// TwinCAT 3 PLC project Untitled1
// ProgramVersion: 3.1.4024.0
// libraries:
//   Tc2_Standard, * (Beckhoff Automation GmbH)
//   Tc2_System, * (Beckhoff Automation GmbH)
//   Tc3_Module, * (Beckhoff Automation GmbH)
//   VisuDialogs, * (System)
//   VisuSymbols,3.5.10.0,System
// project tree:
//   / DUT.TcDUT, GlobalTextList.TcGTLO, Param.TcGVL, PlcTask.TcTTO, Visualization Manager.TcVMO (not stored)
//   DUTs/ weekDays.TcDUT
//   GVLs/ GVL.TcGVL
//   POUs/ MAIN.TcPOU, Routine1.TcPOU, Routine2.TcPOU
//   VISUs/ Visualization.TcVIS
// real-time tasks:
//   TASK PlcTask: cycle T#10ms, priority 20, ADS port 350

CONFIGURATION Untitled1
    RESOURCE PLC ON TwinCAT3
        TASK PlcTask(INTERVAL := T#10ms, PRIORITY := 20);
        PROGRAM MAIN WITH PlcTask : MAIN;
    END_RESOURCE
END_CONFIGURATION

// ---- DUT.TcDUT
TYPE DUT :
STRUCT
END_STRUCT
END_TYPE

// ---- DUTs/weekDays.TcDUT
TYPE weekDays :
STRUCT
	Mon : STRING;
	Tue : STRING;
	Wend: STRING;
	Thu	: STRING;
	Fri	: STRING;
	
END_STRUCT
END_TYPE

// ---- GVLs/GVL.TcGVL
{attribute 'qualified_only'}
VAR_GLOBAL
	Morning 		: BOOL := FALSE	 ;
	
	WakeUp			: BOOL	 ;
	DateCheck		: BOOL	 ;
	ComeBackHome	: BOOL	 ;
	TakeShower		: BOOL	 ;
	GoToBed			: BOOL 	 ;
	MakeTheBed		: BOOL   ;
	MakeCoffee		: BOOL	 ;
	EatBreakfast	: BOOL	 ;
	Day 			: STRING ;
	Routine1 		: BOOL 	 ;
	Routine2		: BOOL	 ;
	
	
			
END_VAR

// ---- Param.TcGVL
{attribute 'qualified_only'}
VAR_GLOBAL CONSTANT
END_VAR

// ---- POUs/MAIN.TcPOU
PROGRAM MAIN
VAR
	State 			: INT	:= 5 ;

	ToTimeoutbool 	: TON ;
	T1Timer 		: BOOL ;
	enable 			: BOOL;
	rTrigenable 	: R_TRIG;
	
END_VAR

rTrigenable(CLk := enable);
ToTimeoutbool(IN := T1Timer,PT := T#2S);
IF gvl.Morning THEN
	state := 0;
END_IF
	CASE state OF
	0:
		GVL.WakeUp 					:= TRUE;
		T1Timer 					:= TRUE;
		IF ToTimeoutbool.Q THEN
			T1Timer 				:= FALSE;
			GVL.WakeUp 				:= FALSE ;
			state := 1; 
		END_IF
		
	1:
		GVL.MakeTheBed 				:= TRUE;
			T1Timer 				:= TRUE;
		IF ToTimeoutbool.Q THEN
			T1Timer 				:= FALSE;
			GVL.MakeTheBed 			:= FALSE ;
			state := 2;
		END_IF
		
	2:
		GVL.TakeShower 				:= TRUE;
		T1Timer 					:= TRUE;
		IF ToTimeoutbool.Q THEN
			T1Timer := FALSE;
			GVL.TakeShower 			:= FALSE ;
			state := 3;
		END_IF
		
	3:
		GVL.DateCheck				:= TRUE;
		State := 4; 

	4: 
		IF gvl.Day = 'Sat' OR gvl.Day = 'Sun' THEN
			routine2();
			gvl.Routine2 			:= TRUE;
			
		ELSIF gvl.Day = 'Fri' OR gvl.Day = 'Mon' OR gvl.Day = 'Tue' OR gvl.Day = 'Wend' OR gvl.Day = 'Thu' THEN
		 	routine1();		
			GVl.Routine1 			:= TRUE ;
			
		END_IF
	
		
	END_CASE

END_PROGRAM

// ---- POUs/Routine2.TcPOU
PROGRAM Routine2
VAR
	     
	DoLaundriesR2             	: BOOL ; 
	DoGroceriesR2            	: BOOL ; 
	
	OrganizeGroceriesR2      	: BOOL ; 
	CheckWashingMachineR2    	: BOOL ; 
	DoOtherChoresR2         	: BOOL ; 
	CookSomethingR2           	: BOOL ; 
	UnloadMachineR2          	: BOOL ;  
	EatLunchR2					: BOOL ;
	State 						: INT :=0  ;
	Day  						: STRING  ;
	ToTimeoutbool 				: TON ;
	T1Timer 					: BOOL ;
	enable 						: BOOL;
	rTrigenable 				: R_TRIG;
END_VAR

rTrigenable(CLk := enable);
ToTimeoutbool(IN := T1Timer,PT := T#2S);
gvl.DateCheck := FALSE ;

CASE state OF
	0:
		GVL.MakeCoffee 					:= TRUE;
		T1Timer 						:= TRUE;
		IF ToTimeoutbool.Q THEN
			T1Timer 					:= FALSE;
			GVL.MakeCoffee 				:= FALSE ;
			state 						:= 1; 
		END_IF
		
	1:
		GVL.EatBreakfast 				:= TRUE;
			T1Timer 					:= TRUE;
		IF ToTimeoutbool.Q THEN
			T1Timer 					:= FALSE;
			GVL.EatBreakfast			:= FALSE ;
			state 						:= 2;
		END_IF
		
	2:
		DoLaundriesR2 					:= TRUE;
			T1Timer 					:= TRUE;
		IF ToTimeoutbool.Q THEN
			T1Timer 					:= FALSE;
			DoLaundriesR2 				:= FALSE ;
			state 						:= 3;
		END_IF
		
	3:
		DoGroceriesR2					:= TRUE;
		T1Timer 						:= TRUE ;
		IF ToTimeoutbool.Q THEN
			T1Timer 					:= FALSE;
			DoGroceriesR2				:= FALSE ;
			state 						:= 4;
		END_IF					
	4: 
		gvl.ComeBackHome				:= TRUE;
		T1Timer 						:= TRUE ;
		IF ToTimeoutbool.Q THEN
			T1Timer 					:= FALSE;
			gvl.ComeBackHome			:= FALSE ;
			state 						:= 5;
		END_IF	
	
	5:
		OrganizeGroceriesR2				:= TRUE;
		T1Timer 						:= TRUE ;
		IF ToTimeoutbool.Q THEN
			T1Timer 					:= FALSE;
			OrganizeGroceriesR2			:= FALSE ;
			state 						:= 6;
		END_IF
	6:
		CheckWashingMachineR2			:= TRUE;
		T1Timer 						:= TRUE ;
		IF ToTimeoutbool.Q THEN
			T1Timer 					:= FALSE;
			CheckWashingMachineR2		:= FALSE ;
			state 						:= 7;
		END_IF
	7:	
		DoOtherChoresR2					:= TRUE;
		T1Timer 						:= TRUE ;
		IF ToTimeoutbool.Q THEN
			T1Timer 					:= FALSE;
			DoOtherChoresR2				:= FALSE ;
			state 						:= 8;
		END_IF
	8:
		CookSomethingR2					:= TRUE;
		T1Timer 						:= TRUE ;
		IF ToTimeoutbool.Q THEN
			T1Timer 					:= FALSE;
			CookSomethingR2				:= FALSE ;
			state 						:= 9;
		END_IF
	9:
		EatLunchR2						:= TRUE;
		T1Timer 						:= TRUE ;
		IF ToTimeoutbool.Q THEN
			T1Timer 					:= FALSE;
			EatLunchR2					:= FALSE ;
			state 						:= 10;
		END_IF
	10:
		UnloadMachineR2					:= TRUE;
		T1Timer 						:= TRUE ;
		IF ToTimeoutbool.Q THEN
			T1Timer 					:= FALSE;
			UnloadMachineR2				:= FALSE ;
			state 						:= 11;
		END_IF
	11:
		GVL.GoToBed						:= TRUE;
		T1Timer 						:= TRUE ;
		IF ToTimeoutbool.Q THEN
			T1Timer 					:= FALSE;
			GVl.GoToBed					:= FALSE ;
			state 						:= 99;
		END_IF

	99:
		gvl.Morning 					:= FALSE;
		
		
END_CASE

END_PROGRAM

// ---- POUs/Routine1.TcPOU
PROGRAM Routine1
VAR
	State 			: INT ;
	ToTimeoutbool 	: TON ;
	T1Timer 		: BOOL ;
	enable 			: BOOL;
	rTrigenable 	: R_TRIG;
	GetReadyR1 		: BOOL ;
	GetIntoCarR1 	: BOOL ;
	GoToworkR1 		: BOOL ;
	
	
	
END_VAR

rTrigenable(CLk := enable);
ToTimeoutbool(IN := T1Timer,PT := T#2S);
gvl.DateCheck := FALSE ;


CASE state OF
	0:
		GVL.MakeCoffee 					:= TRUE;
		T1Timer 						:= TRUE;
		IF ToTimeoutbool.Q THEN
			T1Timer 					:= FALSE;
			GVL.MakeCoffee 				:= FALSE ;
			state 						:= 1; 
		END_IF
		
	1:
		GVL.EatBreakfast 				:= TRUE;
			T1Timer 					:= TRUE;
		IF ToTimeoutbool.Q THEN
			T1Timer 					:= FALSE;
			GVL.EatBreakfast			:= FALSE ;
			state 						:= 2;
		END_IF
		
	2:
		GetReadyR1 						:= TRUE;
		T1Timer 						:= TRUE;
		IF ToTimeoutbool.Q THEN
			T1Timer 					:= FALSE;
			GetReadyR1 					:= FALSE ;
			state 						:= 3;
		END_IF
		
	3:
		GetIntoCarR1					:= TRUE;
		T1Timer 						:= TRUE ;
		IF ToTimeoutbool.Q THEN
			T1Timer 					:= FALSE;
			GetIntoCarR1				:= FALSE ;
			state 						:= 4;
		END_IF					
	4: 
		GoToworkR1						:= TRUE;
		T1Timer 						:= TRUE ;
		IF ToTimeoutbool.Q THEN
			T1Timer 					:= FALSE;
			GoToworkR1					:= FALSE ;
			state 						:= 5;
		END_IF	
	
	5:
		GVL.ComeBackHome				:= TRUE;
		T1Timer 						:= TRUE ;
		IF ToTimeoutbool.Q THEN
			T1Timer 					:= FALSE;
			GVL.ComeBackHome			:= FALSE ;
			state 						:= 6;
		END_IF	
		
	6:
		GVL.GoToBed						:= TRUE;
		T1Timer 						:= TRUE ;
		IF ToTimeoutbool.Q THEN
			T1Timer 					:= FALSE;
			GVL.GoToBed					:= FALSE ;
			state 						:= 7;
		END_IF	
	7:
		gvl.Morning 					:= FALSE;
		
END_CASE

END_PROGRAM

// ---- GlobalTextList.TcGTLO
TEXTLIST GlobalTextList
  898 = 'Check Date'
  423 = 'Check Laundry'
  560 = 'chores'
  648 = 'Come Back Hoem'
  250 = 'Come Back Home'
  218 = 'Common routine'
  574 = 'Common Routine'
  128 = 'Cook'
  342 = 'Eat'
  561 = 'Eat Breakfast'
  868 = 'Enter the date'
  53 = 'Get Into Car'
  382 = 'GetIntoCar'
  387 = 'GetReady'
  285 = 'Go to Bed'
  981 = 'Go to Work'
  411 = 'Groceries'
  69 = 'Label'
  906 = 'Laundry'
  545 = 'Make Bed'
  225 = 'Make Coffee'
  589 = 'organize Groceries'
  904 = 'sat'
  970 = 'Showering'
  175 = 'Start a day'
  536 = 'Unload Washing'
  403 = 'Wake Up'
  576 = 'WakeUp'
  460 = 'Weekdays'
  921 = 'Weekend'
  882 = 'Working Days'
END_TEXTLIST

// ---- VISUs/Visualization.TcVIS
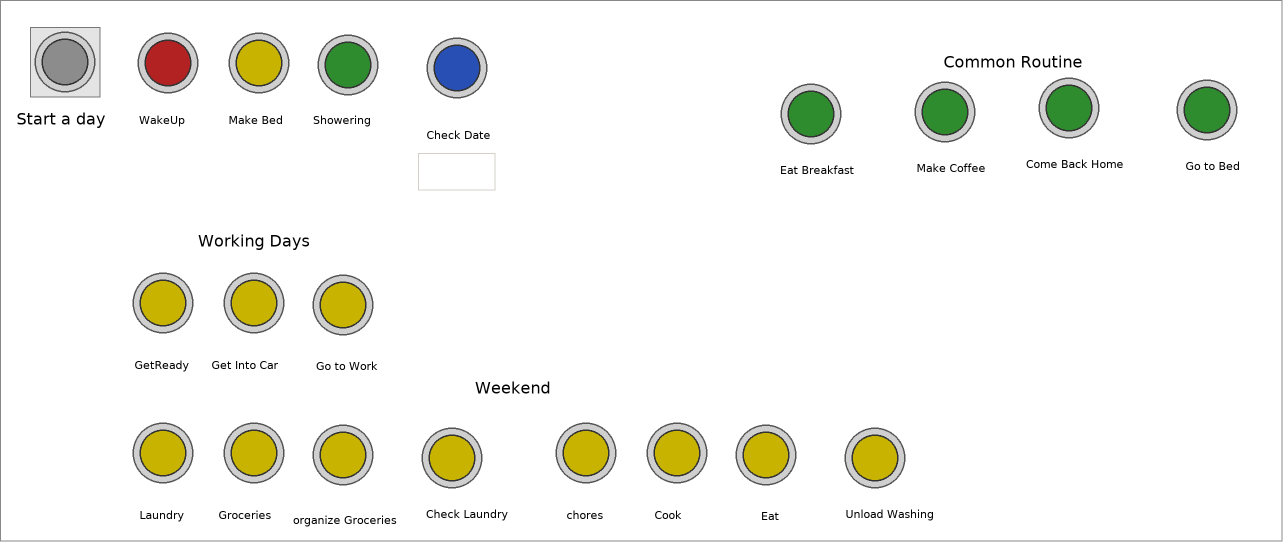
VISUALIZATION Visualization  // 1283x542
    Textfield (418,153 77x37), text variable: GVL.Day
        OnMouseClick: write the text variable via Edit
    Lamp1 (133,28 70x70), variable: gvl.WakeUp, style: Lamp-Lamp1-Red
    Lamp1 (224,28 70x70), variable: gvl.MakeTheBed, style: Lamp-Lamp1-Yellow
    Lamp1 (313,30 70x70), variable: gvl.TakeShower, style: Lamp-Lamp1-Green
    Lamp1 (422,33 70x70), variable: gvl.DateCheck, style: Lamp-Lamp1-Blue
    PushSwitch (30,27 70x70), variable: gvl.Morning, behaviour: TAP, style: Switch-PushSwitch-Gray
    Label (128,103 68x35), "WakeUp"
    Label (420,117 77x37), "Check Date"
    Label (221,103 70x35), "Make Bed"
    Label (308,103 68x35), "Showering"
    Group (128,268 253x116)
        Lamp1 (0,0 70x70), variable: Routine1.GetReadyR1, style: Lamp-Lamp1-Yellow
        Lamp1 (91,0 70x70), variable: Routine1.GetIntoCarR1, style: Lamp-Lamp1-Yellow
        Lamp1 (180,2 70x70), variable: Routine1.GoToworkR1, style: Lamp-Lamp1-Yellow
        Label (0,80 68x35), "GetReady"
        Label (185,81 68x35), "Go to Work"
        Label (83,80 68x35), "Get Into Car"
    Group (128,418 818x124)
        Lamp1 (289,5 70x70), variable: Routine2.CheckWashingMachineR2, style: Lamp-Lamp1-Yellow
        Lamp1 (0,0 70x70), variable: Routine2.DoLaundriesR2, style: Lamp-Lamp1-Yellow
        Lamp1 (91,0 70x70), variable: Routine2.DoGroceriesR2, style: Lamp-Lamp1-Yellow
        Lamp1 (180,2 70x70), variable: Routine2.OrganizeGroceriesR2, style: Lamp-Lamp1-Yellow
        Label (0,80 68x35), "Laundry"
        Label (283,79 112x35), "Check Laundry"
        Label (154,81 126x43), "organize Groceries"
        Label (83,80 68x35), "Groceries"
        Lamp1 (712,5 70x70), variable: Routine2.UnloadMachineR2, style: Lamp-Lamp1-Yellow
        Lamp1 (423,0 70x70), variable: Routine2.DoOtherChoresR2, style: Lamp-Lamp1-Yellow
        Lamp1 (514,0 70x70), variable: Routine2.CookSomethingR2, style: Lamp-Lamp1-Yellow
        Lamp1 (603,2 70x70), variable: Routine2.EatLunchR2, style: Lamp-Lamp1-Yellow
        Label (423,80 68x35), "chores"
        Label (706,79 112x35), "Unload Washing"
        Label (608,81 68x35), "Eat"
        Label (506,80 68x35), "Cook"
    Group (761,73 508x115)
        Lamp1 (149,4 70x70), variable: GVL.MakeCoffee, style: Lamp-Lamp1-Green
        Label (134,78 112x35), "Make Coffee"
        Lamp1 (15,6 70x70), variable: GVL.EatBreakfast, style: Lamp-Lamp1-Green
        Label (0,80 112x35), "Eat Breakfast"
        Lamp1 (273,0 70x70), variable: GVL.ComeBackHome, style: Lamp-Lamp1-Green
        Label (258,74 112x35), "Come Back Home"
        Lamp1 (411,2 70x70), variable: GVL.GoToBed, style: Lamp-Lamp1-Green
        Label (396,76 112x35), "Go to Bed"
    Label (179,226 150x30), "Working Days"
    Label (938,47 150x30), "Common Routine"
    Label (438,373 150x30), "Weekend"
    Label (-14,104 150x30), "Start a day"
END_VISUALIZATION
